RESOURCE_TYPE _CBCoreSingle
  (* Standard: 61499-2 *)
  (* Version 0.1, 2019-00-29, hpea485, UOA *)
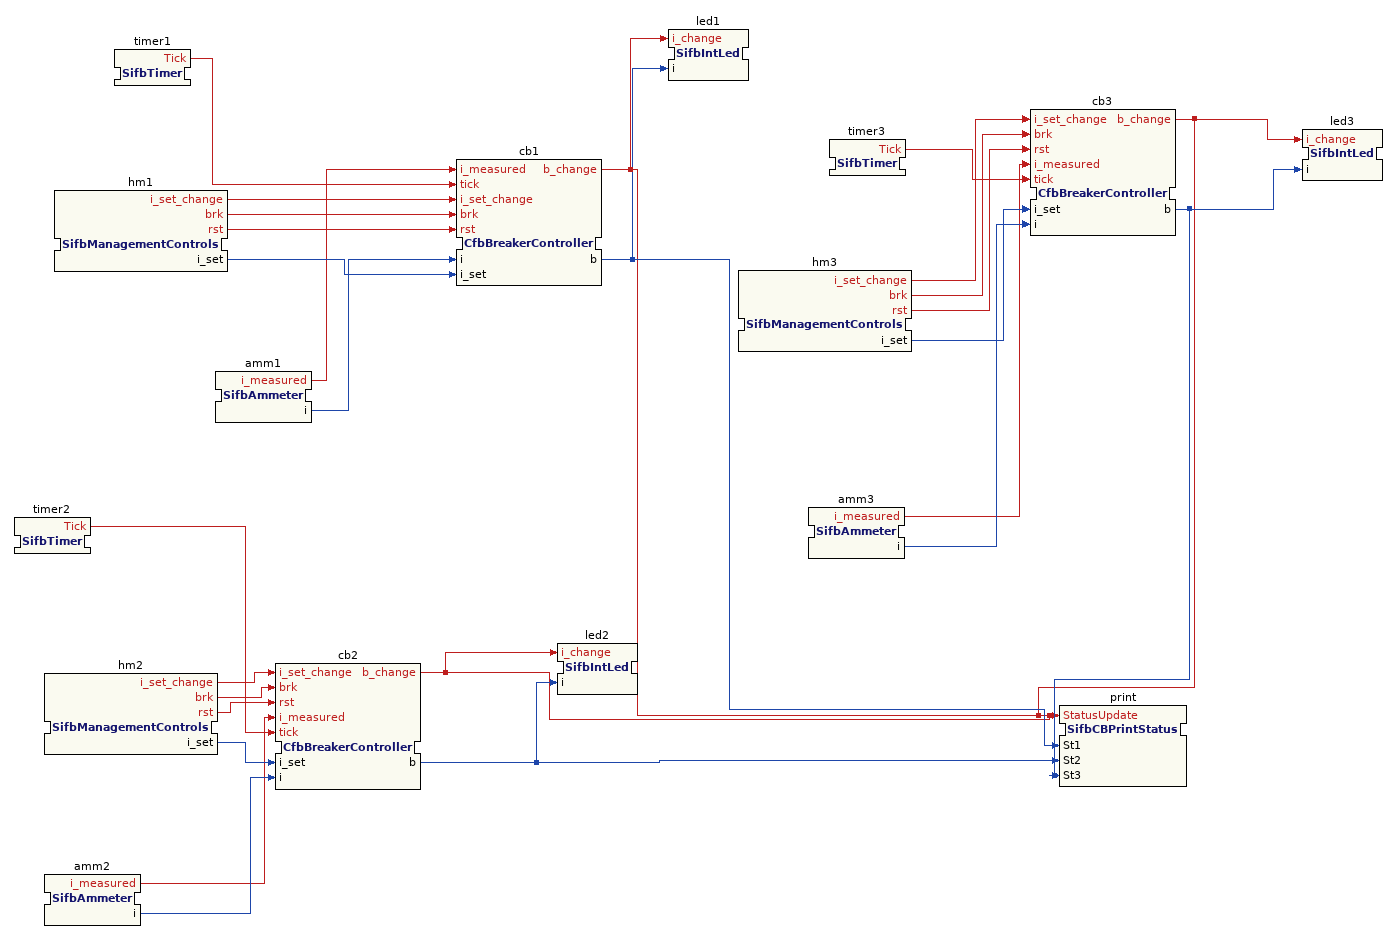
  FBS
    amm1 : SifbAmmeter;
    timer1 : SifbTimer;
    cb1 : CfbBreakerController;
    hm1 : SifbManagementControls;
    led1 : SifbIntLed;
    hm3 : SifbManagementControls;
    led3 : SifbIntLed;
    amm3 : SifbAmmeter;
    cb3 : CfbBreakerController;
    timer3 : SifbTimer;
    hm2 : SifbManagementControls;
    led2 : SifbIntLed;
    amm2 : SifbAmmeter;
    cb2 : CfbBreakerController;
    timer2 : SifbTimer;
    print : SifbCBPrintStatus;
  END_FBS
  EVENT_CONNECTIONS
    amm1.i_measured TO cb1.i_measured;
    timer1.Tick TO cb1.tick;
    cb1.b_change TO led1.i_change;
    cb1.b_change TO print.StatusUpdate;
    hm1.i_set_change TO cb1.i_set_change;
    hm1.brk TO cb1.brk;
    hm1.rst TO cb1.rst;
    hm3.i_set_change TO cb3.i_set_change;
    hm3.brk TO cb3.brk;
    hm3.rst TO cb3.rst;
    amm3.i_measured TO cb3.i_measured;
    cb3.b_change TO led3.i_change;
    cb3.b_change TO print.StatusUpdate;
    timer3.Tick TO cb3.tick;
    hm2.i_set_change TO cb2.i_set_change;
    hm2.brk TO cb2.brk;
    hm2.rst TO cb2.rst;
    amm2.i_measured TO cb2.i_measured;
    cb2.b_change TO led2.i_change;
    cb2.b_change TO print.StatusUpdate;
    timer2.Tick TO cb2.tick;
  END_CONNECTIONS
  DATA_CONNECTIONS
    amm1.i TO cb1.i;
    cb1.b TO led1.i;
    cb1.b TO print.St1;
    hm1.i_set TO cb1.i_set;
    hm3.i_set TO cb3.i_set;
    amm3.i TO cb3.i;
    cb3.b TO led3.i;
    cb3.b TO print.St3;
    hm2.i_set TO cb2.i_set;
    amm2.i TO cb2.i;
    cb2.b TO led2.i;
    cb2.b TO print.St2;
  END_CONNECTIONS
END_RESOURCE_TYPE
